TEXTLIST TaschenrechnerBefehle
  0 = '-'
  1 = 'usint addieren (unsigned short int; 8 bit)'
  2 = 'sint addieren (signed short int; 8 bitI)'
   = ''
END_TEXTLIST

(* stored: Version 1.1.0.1, ProductVersion 3.1.4022.6
   TextList TaschenrechnerBefehle: Id {6bf491f1-6666-4c6d-aec4-8eb0ef784ca6} *)
